// TIA Portal V19 export
DATA_BLOCK "A04_0304TrkManager"   // DB184
// stored: InstanceOfName A04_0304TrkManager_FB, InstanceOfType FB
"A04_0304TrkManager_FB"
   // VAR_INPUT
   //    AreaInterface : "AreaInterface";
   //    SuperUserLogged : Bool;
   // END_VAR
   // VAR
   //    HMI : Struct
   //       Move { S7_SetPoint := 'True'} : Array[1..20] of "TrkMng_Move";
   //       NumDelete { S7_SetPoint := 'True'} : Int;
   //    END_STRUCT;
   //    Sts : Struct
   //       Move : Struct
   //          SelectionOn : Bool;
   //          SelectionNo : Int;
   //       END_STRUCT;
   //    END_STRUCT;
   //    TON_Delete_Buttons : IEC_TIMER;
   // END_VAR
BEGIN
END_DATA_BLOCK
